FUNCTION_BLOCK FB_SUB_LREAL_ARR96 (* Subtracts two LREAL arrays of size 96 *)
  (* Standard: 61499-1; Classification: Mathematic; Function: SUBTRACTOR; Type: Mathematical function; Description: Derived from FB_SUB_LREAL. Subtracts two arrays of size [96] from one another. *)
  (* Version 1.0, 2007-06-26, TS, PROFACTOR GmbH *)
  (* Version 1.1, 2017-05-16, Marc Jakobi, HTW Berlin, Adjusted FB_SUB_LREAL for arrays of size 96 *)
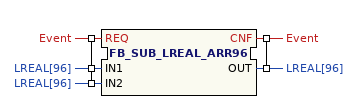
  EVENT_INPUT
    REQ WITH IN1, IN2; (* Normal Execution Request *)
  END_EVENT
  EVENT_OUTPUT
    CNF WITH OUT; (* Execution Confirmation *)
  END_EVENT
  VAR_INPUT
    IN1 : ARRAY [0..95] OF LREAL; (* First funtion input *)
    IN2 : ARRAY [0..95] OF LREAL; (* Second function input *)
  END_VAR
  VAR_OUTPUT
    OUT : ARRAY [0..95] OF LREAL; (* Function output *)
  END_VAR
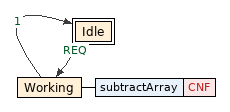
  EC_STATES
    Idle; (* Initial State *)
    Working : subtractArray -> CNF; (* Normal execution *)
  END_STATES
  EC_TRANSITIONS
    Idle TO Working := REQ;
    Working TO Idle := 1;
  END_TRANSITIONS
  ALGORITHM subtractArray IN ST: (* Normally executed algorithm *)
VAR
	i : UINT;
END_VAR
FOR i := 0 TO 95 BY 1 DO
	OUT[i] := IN1[i] - IN2[i];
END_FOR;
  END_ALGORITHM
END_FUNCTION_BLOCK
